// Mitsubishi GX Works2 project: 0710-z0   PLC: Q02/Q02H

PROGRAM MAIN
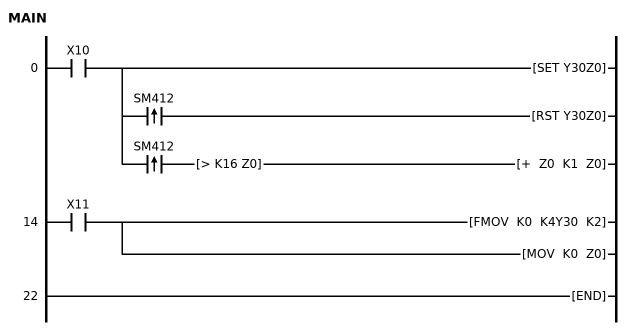
0     LD      X10
      SET     Y30Z0
      MPS
      ANDP    SM412
      RST     Y30Z0
      MPP
      ANDP    SM412
      AND>    K16 Z0
      +       Z0 K1 Z0
14    LD      X11
      FMOV    K0 K4Y30 K2
      MOV     K0 Z0
22    END
END_PROGRAM
